PROGRAM Automatic_Or_Manual
VAR_INPUT
	Automatic_Or_Manual:BOOL;
END_VAR

IF Automatic_Or_Manual THEN
	Automatic();
ELSE
	Manual();
END_IF

END_PROGRAM

(* stored: Version 1.1.0.1, ProductVersion 3.1.4024.12
   POU Automatic_Or_Manual: Id {eb7c2b8b-a0a7-45e5-82a9-2d4c86ed9423}, SpecialFunc None *)
